// TIA Portal V19 export
DATA_BLOCK "Area02_HU"   // DB127
// stored: InstanceOfName Area02_HU_FB, InstanceOfType FB
"Area02_HU_FB"
   // VAR_INPUT
   //    AreaInterface : "AreaInterface";
   // END_VAR
   // VAR_OUTPUT
   //    MachineInterface : "MachineInterface";
   // END_VAR
   // VAR
   //    Pump : "HU_Pump";
   //    Tank { S7_SetPoint := 'True'} : "HU_Tank";
   //    HMI : Struct
   //       Pressure_FinalCut : Real;
   //    END_STRUCT;
   // END_VAR
BEGIN
END_DATA_BLOCK
